// TIA Portal V19 export
TYPE "LAF_typeDevDiagStatesMode"
TITLE = Structure device diag state mode / Struktur Status Mode
// This data type contains the structure of the parameter and return values of the devices. / PN device Diagnose
// stored: Access Published
   STRUCT
      laddr { ExternalAccessible := 'False'; ExternalVisible := 'False'; ExternalWritable := 'False'} : HW_IOSYSTEM;   // Local Adress
      mode { ExternalAccessible := 'False'; ExternalVisible := 'False'; ExternalWritable := 'False'} : UInt;   // Mode 1..5
      retVal { ExternalAccessible := 'False'; ExternalVisible := 'False'; ExternalWritable := 'False'} : Int;   // Rückmeldung / Return Value
      state { ExternalAccessible := 'False'; ExternalVisible := 'False'; ExternalWritable := 'False'} : Array[0..1024] of Bool;   // Array 0..1024
   END_STRUCT;
END_TYPE
